INTERFACE I_WashStrategy

METHOD GetDuration
VAR_INPUT
END_VAR
END_METHOD

METHOD Start
VAR_INPUT
END_VAR
END_METHOD

METHOD Stop
VAR_INPUT
END_VAR
END_METHOD

END_INTERFACE

(* stored: Version 1.1.0.1, ProductVersion 3.1.4024.16
   Itf I_WashStrategy: Id {6c2c2703-ab12-4238-99e3-cc10feaf744e}
   Method GetDuration: Id {4f214b80-74b8-4b0b-a1e0-7484f2ccb3ff}
   Method Start: Id {8dab1351-8746-429b-81bf-0dda65a2482f}
   Method Stop: Id {08bd247e-b3d3-42fe-b628-1d39af0f0cac} *)
